FUNCTION F_SensorLog : BOOL
VAR_INPUT
	iLevel: INT;
	sName : STRING;
	bNew  : BOOL;
END_VAR
VAR
	
END_VAR
VAR_IN_OUT
	bOld : BOOL;
END_VAR

IF (bOld <> bNew) THEN
	Logging.fbSensorLog.P_sModule := 'IO Toggled';
	Logging.fbSensorLog.M_nLogger(iLogLevel:= Logging.fbDebugLog.P_iLogVerbosity, 
								sSource:= sName , sMessage:=  F_Concat3(BOOL_TO_STRING(bOld),'->',BOOL_TO_STRING(bNew)));
							// sMessage:=  F_Concat5(sName, ',', BOOL_TO_STRING(bOld),'->',BOOL_TO_STRING(bNew)));
	bOld := bNew;
END_IF

END_FUNCTION

(* stored: Version 1.1.0.1, ProductVersion 3.1.4022.18
   POU F_SensorLog: Id {b505390a-e997-43b2-a731-7ed5f7b4f3bd}, SpecialFunc None *)
